{attribute 'qualified_only'}
{attribute 'strict'}
TYPE E_MAIN_STATE_MACHINE :
(
    INIT := 0,
    NOMINAL := 1,
    EXCHANGE_MODE := 2,
    BUTTON_WAIT := 3

);
END_TYPE

(* stored: Version 1.1.0.1, ProductVersion 3.1.4024.12
   DUT E_MAIN_STATE_MACHINE: Id {04c7a38b-f2a2-42a7-8850-fcc470324d66} *)
